# EPICS substitutions: ffmpegServerApp/Db/pluginMJPG.substitutions
#
# pluginMJPG.substitutions
#

file NDPluginBase.template
{
	{
	P				=	$(CAM):,
	R				=	MJPG$(N):,
	PORT			=	MJPG$(N),
	ADDR			=	"\$(ADDR=0)",
	TIMEOUT			=	"\$(TIMEOUT=1)",
	NDARRAY_PORT	=	$(PLUGIN_SRC),
	NDARRAY_ADDR	=	0,
	BIT_DEPTH		=	$(IMAGE_BIT_DEPTH),
	}
}

# Macros:
#  P        Device Prefix
#  R        Device Suffix
#  PORT     Asyn Port name
#  QUALITY  Jpeg Quality in percent
#  MAXW     Maximum Jpeg Width
#  MAXH     Maximum Jpeg Height
file ffmpegStream.template
{
	{
	P				=	$(CAM):,
	R				=	MJPG$(N):,
	PORT			=	MJPG$(N),
	ADDR			=	"\$(ADDR=0)",
	TIMEOUT			=	"\$(TIMEOUT=1)",
	QUALITY			=	100,
	}
}
